FUNCTION_BLOCK FB_RobotRegionMove_FeedInConveyor_V2 EXTENDS FB_ObjectBase_V2 IMPLEMENTS IBasicElement
VAR_INPUT
    Robot     					: REFERENCE TO FB_FanucRobot_Basic_V2;
	LowerConveyor				: REFERENCE TO FB_Motor;
	Input 						: REFERENCE TO ST_InputTable;

   // Command   : ST_WareHouseWithRobotMove_Command;
    Info	  					: ST_RobotRegionMove_Info;
	Stop	  					: BOOL;
	bCheckUpperCV_ServiceDone	: BOOL;
END_VAR
VAR_OUTPUT
  // Status : ST_WareHouseWithRobotMove_Status;
  
END_VAR
VAR
	//_Abort		: BOOL;
	strStatus	: STRING;
	uiResumeStep : UDINT;
	
	Area	: E_RobotArea := E_RobotArea.InOutConveyor;
	UseA 	: BOOL;
	UseB	: BOOL;
	
	Get 	:BOOL;
	tonTimeOut	:TON;
	bTimeOutIN			   : BOOL;
	tonDelay	 : TON;
	_UniqueErrorCode :STRING;
	PreviousStrStatus : STRING;
	PreviousErrorCode : STRING;
	//Added by Jidien Kachu in 2025/10/09
	uiLastBothStep	: UINT;
	uiLastSingleClampStep	: UINT;
	bRobotTimeOutIN	: BOOL;
	tonRobotTimeOut	: TON;
	uiBothStep	: UINT;
	uiSingleClampStep	: UINT;	
	
	_bRetry	: BOOL;
END_VAR

SUPER^.A10_StateControl();
A00_BasicUnits();

(*============================================================
Create Date : 2025/11/24
Last Update	: 2026/04/01
Change Log  : 2025/11/24，Fix StateControl Switch , the version extend Kachue verion from TH_Mirror DAS // Edited : Gamin
			  2026/04/01，移植泰興鏡射機版本。
============================================================*)

ACTION A00_BasicUnits:
tonTimeOut(IN:= bTimeOutIN AND NOT THIS^.Stop, PT:=T#60S);
tonDelay(PT:=T#1S);
tonRobotTimeOut(IN:= bRobotTimeOutIN AND NOT THIS^.Stop, PT:=T#60S);
ErrorID:=2240;
END_ACTION

METHOD M_CheckCommand : BOOL // True : Command is useful
VAR_INPUT
END_VAR
VAR
	
END_VAR
// Check command paremeter is correct
	
	THIS^.Get :=Info.Get;
	UseA := Info.UseA;
	UseB := Info.UseB;

	 //FeedIn/Out conveyor
	 	IF UseA THEN	 
			IF  (Info.A_Position<1 OR  Info.A_Position>3 )THEN
				strStatus:='Wrong command ,Position A Not allow';
				M_CheckCommand:=FALSE;
				RETURN;	
			ELSIF  Info.A_Position=3 AND Get THEN
				strStatus:='Wrong command ,Can Not Get box from FeedOut conveyor ';
				M_CheckCommand:=FALSE;
				RETURN;
			ELSIF 	Info.A_Position <>3 AND NOT Get THEN
				strStatus:='Wrong command ,Can Not Put box to FeedIn conveyor ';
				M_CheckCommand:=FALSE;
				RETURN;				
			END_IF
		END_IF
		
		IF UseB AND ( Info.B_Position<1 OR  Info.B_Position>3 )THEN
			strStatus:='Wrong command ,Position B Not allow';
			M_CheckCommand:=FALSE;
			RETURN;	
		ELSIF UseB AND Info.B_Position=3 AND Get THEN
			strStatus:='Wrong command ,Can Not Get box from FeedOut conveyor ';
			M_CheckCommand:=FALSE;
			RETURN;		
		ELSIF UseB AND Info.B_Position <>3 AND NOT Get THEN
			strStatus:='Wrong command ,Can Not Put box to FeedIn conveyor ';
			M_CheckCommand:=FALSE;
			RETURN;		
		END_IF
		
M_CheckCommand:=TRUE;
END_METHOD

METHOD M_CheckUnitsNotBusy : BOOL
VAR_INPUT
END_VAR
M_CheckUnitsNotBusy := true;
END_METHOD

METHOD M_CheckUnitsReady : BOOL
VAR_INPUT
END_VAR
M_CheckUnitsReady := true;
END_METHOD

METHOD M_ResetHomingFeedOut : BOOL
VAR_INPUT
END_VAR
Execute := FALSE;
info.UseA := FALSE;
info.UseB := FALSE;

M_ResetHomingFeedOut := TRUE;
END_METHOD

METHOD M_StartHomingFeedOut : BOOL
VAR_INPUT
	UseA	: BOOL;
	UseB	: BOOL;
END_VAR
// NG conveyor homing only place
Info.Get := FALSE;

Info.UseA := UseA;
info.UseB := UseB;

IF UseA AND UseB THEN
	Info.A_Position := 3;
	Info.B_Position := 3;
ELSIF UseA THEN
	Info.A_Position := 3;
	info.B_Position := 99;
ELSIF UseB THEN
	info.A_Position	:= 99;
	Info.B_Position := 3;
END_IF

Execute := TRUE;

M_StartHomingFeedOut := TRUE;
END_METHOD

METHOD  M_STATE_ABORTED
VAR_INPUT
END_VAR
IF NOT _bRetry THEN
	Busy	:= FALSE;
	Error 	:= TRUE;
	Aborted := TRUE;
	Status 	:= strStatus;
	UniqueErrorCode:=_UniqueErrorCode;
	uiAbortingStep := 0;
	_AbortCompleted:=FALSE;//Edited by Jidien Kachu in 2025/10/14
END_IF

IF reset THEN
	_bRetry := TRUE;
	Error 	:= FALSE;
	Aborted := FALSE;
END_IF

IF NOT Execute THEN
	eSTATE:=STATE_RESETTING;
END_IF
IF Execute AND _bRetry AND NOT Robot._DI1.Error AND NOT Robot.Halt THEN
	PreviousStrStatus := strStatus;
	PreviousErrorCode := _UniqueErrorCode;
	uiExecutingStep   := uiResumeStep;
	(* Edited by Jidien Kachu in 2025/10/09 *)
	uiBothStep 		  := uiLastBothStep;
	uiSingleClampStep := uiLastSingleClampStep;

	Status := '';

	(*====================================*)
	IF GVL_ADS.MachineState <>E_MachineState.Error THEN
		eSTATE:=STATE_EXECUTING;
	END_IF
END_IF
END_METHOD

METHOD  M_STATE_ABORTING
VAR_INPUT
END_VAR
CASE uiAbortingStep OF
	0 :
			bTimeOutIN		:= FALSE;
			bRobotTimeOutIN := FALSE;
			tonDelay.IN 	:= FALSE;
			_bRetry:= FALSE;
			_Abort := FALSE;
			
			LowerConveyor.M_MotorStop();
			IF strStatus = PreviousStrStatus THEN
				_UniqueErrorCode :=PreviousErrorCode;
			END_IF
			uiAbortingStep:=100;
	100:		
			 IF DAS_CoreSys.MachineControl.M_RobotResetCmd() THEN
				 uiAbortingStep := 200;
			 END_IF
	200:
			IF DAS_CoreSys.MachineControl.M_RobotStartCmd() THEN
				 uiAbortingStep := 300;
			 END_IF 
	300:
			IF Robot._DI1.Error THEN
		 		uiAbortingStep := 100;
			ELSE
				uiAbortingStep := 9999;
			END_IF
	
	9999:	
			_AbortCompleted:=TRUE;
END_CASE

IF _AbortCompleted THEN	
	eSTATE :=STATE_ABORTED;
END_IF
END_METHOD

METHOD  M_STATE_DONE
VAR_INPUT
END_VAR
Busy := FALSE;
Done := TRUE;
IF NOT Execute THEN
    eState := STATE_RESETTING;
END_IF
END_METHOD

METHOD  M_STATE_DORMANT
VAR_INPUT
END_VAR
// Clear FB output
Busy            := FALSE;
Done            := FALSE;
_Abort			:= FALSE;
Aborted         := FALSE;
Error           := FALSE;
ErrorID         := 0;
Status          := '';
_ResetCompleted := FALSE;
_Error          := FALSE;
_Executed       := FALSE;
tonDelay.IN := FALSE;
bTimeOutIN:=FALSE;
bRobotTimeOutIN := FALSE;
strStatus :='No Error';
uiExecutingStep :=uiResettingStep :=uiResumeStep :=0;
uiBothStep			:= 0; 
uiSingleClampStep 	:= 0;
uiLastBothStep		:= 0; 
uiLastSingleClampStep := 0; 
_UniqueErrorCode :='0';
tonRobotTimeOut.IN := FALSE;
PreviousStrStatus			 :='';
PreviousErrorCode			 :='';
_bRetry				:= FALSE;

// Wait Execute command
IF Execute AND NOT stop THEN
    eState := STATE_EXECUTING;
END_IF
END_METHOD

METHOD  M_STATE_ERROR
VAR_INPUT
END_VAR
ERROR   :=TRUE;
Busy	:=FALSE;
Status := strStatus;
UniqueErrorCode:=_UniqueErrorCode;
IF NOT Execute THEN	
eSTATE:=STATE_RESETTING;
END_IF
END_METHOD

METHOD  M_STATE_EXECUTING
VAR_INPUT
END_VAR
VAR_INST
	BoxReady_1st : BOOL;
	BoxReady_2nd : BOOL;
//    uiBothStep : UINT;
//    uiSingleClampStep : UINT;	
	Address_A : INT;
	Address_B : INT;
END_VAR
VAR
	WareHouse: INT;
END_VAR
// Set Busy active edit by johnson
Busy := TRUE;
(*IF THIS^.Stop THEN // Pending the timeout when Stop signal occur
	bTimeoutIN:=FALSE;
END_IF*)
// Service Process
CASE uiExecutingStep OF
	0:
        // Clear variable
//        uiBothStep := 0;
		uiLastBothStep := 0; //Edited by Jidien Kachu in 2025/10/09
//		uiSingleClampStep :=0;
		uiLastSingleClampStep := 0; //Edited by Jidien Kachu in 2025/10/09
		BoxReady_1st := 0;
		BoxReady_2nd := 0;
		bTimeOutIN:=FALSE;
        // Check command
        IF M_CheckCommand() THEN
            uiExecutingStep := 10;
		ELSE
			_Error:=TRUE;
        END_IF
    10:
        // Start process, check units first
        IF M_CheckUnitsReady() THEN
            uiExecutingStep := 20;
        END_IF
    20:
        // CHeck units not busy state
        IF M_CheckUnitsNotBusy() THEN
            uiExecutingStep := 1000;
        END_IF
   
	1000:   
			// Read   coordinate
			 Area := THIS^.Area;
 			 Address_A := LREAL_TO_INT(Info.A_Position);
			 Address_B := LREAL_TO_INT(Info.B_Position);
			 
			IF UseA AND NOT UseB THEN
				//Only clampA
				uiExecutingStep := 10000;
			ELSIF NOT UseA AND UseB THEN
				//Only ClampB 
				uiExecutingStep := 20000;
			ELSIF UseA AND UseB THEN
				//Both Clamps
				uiExecutingStep := 30000;		
			ELSE
				strStatus := 'FB_RobotRegionMove_FeedInConveyor_V2 Step 1000: No clamp selected';
				_Error 	  := TRUE;
			END_IF

	10000:	// 檢查 A爪 Sensor判斷是否可以安全做動
			IF Get THEN
				IF  Robot._DI1.ClampA_Open THEN		// AClamp has box
					uiExecutingStep := 11000;
				ELSE
					_Error 	  := TRUE;
					strStatus := 'FB_RobotRegionMove_FeedInConveyor_V2 Step 10000: AClamp not open';
				END_IF
			ELSE
				IF NOT Robot._DI1.ClampA_Open THEN	// AClamp has box
					uiExecutingStep := 11000;
				ELSE	
					_Error 	  := TRUE;
					strStatus := 'FB_RobotRegionMove_FeedInConveyor_V2 Step 10000: AClamp is open';
				END_IF
			END_IF
       
    11000: // Only ClampA 
        IF NOT Robot._DI1.Done THEN
            
            
			CASE uiSingleClampStep OF
				
				0://
				
					CASE Address_A OF
						1,2:
							uiSingleClampStep:=1000;
						
						3: 
							uiSingleClampStep:=100;
					END_CASE
				
				100:	
					LowerConveyor.M_MoveBackward();
					tonDelay.IN := FALSE;
					IF ( NOT Input.bLowCV_BoxArrived_Sensor) AND ( Input.bLowCV_2ndBoxGap_Sensor) THEN
						bTimeOutIN:=FALSE;
						uiSingleClampStep:=150;
					END_IF
					bTimeOutIN:=TRUE;
					IF tonTimeOut.Q=TRUE OR Robot._DI1.Error THEN
						strStatus := 'FB_RobotRegionMove_FeedInConveyor_V2 Step 11000: Empty conveyor timeout';
						uiResumeStep:=11000;
						uiLastSingleClampStep := 0; //Edited by Jidien Kachu in 2025/10/09
						uiAbortingStep := 0;//Edited by Jidien Kachu in 2025/10/14
						_Abort:=TRUE;
					END_IF
				150:
					tonDelay.IN := TRUE;
					IF tonDelay.Q THEN
						uiSingleClampStep:=200;
					END_IF	
				200:
					tonDelay.IN := FALSE;
					LowerConveyor.M_MotorStop();
					uiSingleClampStep:=300;
				
				300:
					IF 	LowerConveyor.InStopped THEN
						bTimeOutIN:=FALSE;
						BoxReady_1st:=TRUE;
						uiSingleClampStep:=9999;
					END_IF
					bTimeOutIN:=TRUE;
					IF tonTimeOut.Q=TRUE OR Robot._DI1.Error THEN
						strStatus :='FB_RobotRegionMove_FeedInConveyor_V2 Step 11000: Stop Conveyor timeout';


						(* Edited by Jidien Kachu in 2025/10/09*)
//						_Error:=TRUE;
						uiResumeStep:=11000;
						uiLastSingleClampStep := 200;
						uiAbortingStep := 0;//Edited by Jidien Kachu in 2025/10/14
						_Abort:=TRUE;
						(*===================================*)
					END_IF	
				
				1000:
						CASE Address_A OF
						1:
								IF 	bCheckUpperCV_ServiceDone THEN
							BoxReady_1st:=Input.bUpCV_Block1Detect_Sensor;
								END_IF
						2:
								IF 	bCheckUpperCV_ServiceDone THEN
							BoxReady_1st:=Input.bUpCV_BoxArrived_Sensor;
								END_IF
						END_CASE						
						
				9999: //
						;
			END_CASE
			          		 
				  // Robot Abs move
           		 Robot.M_StartRobotAbsMove(GetBox:=Get,
											UseClampA:=UseA,
											UseClampB:=UseB,
											Area:=Area,
											ClampA_Address:=Address_A,
											ClampB_Address:=Address_B,
											BoxReady_1:=BoxReady_1st,
											BoxReady_2:=BoxReady_2nd);				  
		
        ELSE
//			bTimeOutIN:=FALSE;
			bRobotTimeOutIN := FALSE; //edited by Jidien Kachu in 2025/10/09
            uiExecutingStep := 10080;
        END_IF
		(* Edited by Jidien Kachu in 2025/10/09*)

		bRobotTimeOutIN := TRUE;

		IF tonRobotTimeOut.Q THEN

			bRobotTimeOutIN := FALSE;
			uiResumeStep 	:= 11000;
			strStatus 		:= 'FB_RobotRegionMove_FeedInConveyor_V2 Step 11000: Robot Abs move timeout';
			_Abort			:= TRUE;
		END_IF	
		IF Robot.Error THEN
			bRobotTimeOutIN := FALSE;
			uiResumeStep 	:= 11000;
			strStatus 		:= CONCAT('FB_RobotRegionMove_FeedInConveyor_V2',robot.ErrMsg);
			_Abort			:= TRUE;
		END_IF
		(*===================================*)
    10080:
        Robot.M_ResetRobotAbsMove(UseA,UseB); // Clear command and go to place box

		bRobotTimeOutIN := TRUE; //Edited by Jidien Kachu in 2025/10/09
        IF NOT Robot._DI1.Done THEN

			bRobotTimeOutIN := FALSE; //Edited by Jidien Kachu in 2025/10/09
            uiExecutingStep := 80000; 
        END_IF
		(* Edited by Jidien Kachu in 2025/10/09 *)

		IF tonRobotTimeOut.Q THEN
			bRobotTimeOutIN := FALSE;
			strStatus 		:= 'FB_RobotRegionMove_FeedInConveyor_V2 Step 10080: Reset Robot timeout';
			_Error:=TRUE;
		END_IF	
		(*=====================================*)
    
	10090: // Check box 

	20000:	// 檢查 B爪 Sensor判斷，是否可以安全做動。
			IF Get THEN
				IF  Robot._DI1.ClampB_Open THEN	// BClamp has box
					uiExecutingStep := 21000;
				ELSE
					_Error	  := TRUE;
					strStatus := 'FB_RobotRegionMove_FeedInConveyor_V2 Step 20000: BClamp not open';
				END_IF
			ELSE
				IF NOT Robot._DI1.ClampB_Open THEN	// BClamp has box
					uiExecutingStep := 21000;
				ELSE
					_Error	  := TRUE;
					strStatus := ' FB_RobotRegionMove_FeedInConveyor_V2 Step 20000: BClamp is open';
				END_IF
			END_IF
		
			
    21000: // Only ClampB
        IF NOT Robot._DI1.Done THEN
			
            	CASE uiSingleClampStep OF
				
				0://
				
					CASE Address_B OF
						1,2:
							uiSingleClampStep:=1000;
						
						3: 
							uiSingleClampStep:=100;
					END_CASE
			
				100:	
					LowerConveyor.M_MoveBackward();
					IF (NOT Input.bLowCV_BoxArrived_Sensor) AND  Input.bLowCV_2ndBoxGap_Sensor THEN
						bTimeOutIN:=FALSE;
						tonDelay.IN := FALSE;
						uiSingleClampStep:=150;
					END_IF
					bTimeOutIN:=TRUE;
					IF tonTimeOut.Q=TRUE OR Robot._DI1.Error THEN
						strStatus 				:= 'FB_RobotRegionMove_FeedInConveyor_V2 Step 21000: Empty conveyor timeout';
						uiResumeStep			:= 21000;
						uiLastSingleClampStep 	:= 0; //Edited by Jidien Kachu in 2025/10/09
						uiAbortingStep 			:= 0;//Edited by Jidien Kachu in 2025/10/14
						_Abort					:= TRUE;
					END_IF
					
				150:
					tonDelay.IN := TRUE;
					IF tonDelay.Q THEN
						uiSingleClampStep:=200;
					END_IF		
				200:
					tonDelay.IN := FALSE;
					LowerConveyor.M_MotorStop();
					uiSingleClampStep:=300;
				
				300:
					IF 	LowerConveyor.InStopped THEN
						bTimeOutIN:=FALSE;
						BoxReady_2nd:=TRUE;
						uiSingleClampStep:=9999;
					END_IF
					bTimeOutIN:=TRUE;
					IF tonTimeOut.Q=TRUE OR Robot._DI1.Error THEN
						strStatus :='FB_RobotRegionMove_FeedInConveyor_V2 Step 21000: Stop Conveyor timeout';




//						_Error:=TRUE;
						(* Edited by Jidien Kachu in 2025/10/09 *)
						uiResumeStep := 21000;
						uiLastSingleClampStep := 200;
						uiAbortingStep := 0;//Edited by Jidien Kachu in 2025/10/14
						_Abort := TRUE;
						(*====================================*)
					END_IF	
				
				1000:

						CASE Address_B OF
						1:
							IF 	bCheckUpperCV_ServiceDone THEN
								BoxReady_2nd:=Input.bUpCV_Block1Detect_Sensor;
							END_IF
													
						2:
							IF 	bCheckUpperCV_ServiceDone THEN
								BoxReady_2nd:=Input.bUpCV_BoxArrived_Sensor;
							END_IF

						END_CASE						
						
				9999 ://
			END_CASE	
		
			
			          		 
				  // Robot Abs move
           		 Robot.M_StartRobotAbsMove( GetBox:=Get,
											UseClampA:=UseA,
											UseClampB:=UseB,
											Area:=Area,
											ClampA_Address:=Address_A,
											ClampB_Address:=Address_B,
											BoxReady_1:=BoxReady_1st,
											BoxReady_2:=BoxReady_2nd);	
        ELSE
//			bTimeOutIN:=FALSE;
			bRobotTimeOutIN := FALSE; //Edited by Jidien Kachu in 2025/10/09
            uiExecutingStep := 20080;
        END_IF
		(* Edited by Jidien Kachu in 2025/10/09 *)

		bRobotTimeOutIN := TRUE;

		IF tonRobotTimeOut.Q THEN

			bRobotTimeOutIN := FALSE;
			uiResumeStep 	:= 21000;
			strStatus 		:= 'FB_RobotRegionMove_FeedInConveyor_V2 Step 21000: Robot Abs move timeout';
			_Abort			:= TRUE;
		END_IF	
		IF Robot.Error THEN
			bRobotTimeOutIN := FALSE;
			uiResumeStep 	:= 21000;
			strStatus 		:= CONCAT('FB_RobotRegionMove_FeedInConveyor_V2',robot.ErrMsg);
			_Abort			:= TRUE;
		END_IF
		(*====================================*)
    20080:
       Robot.M_ResetRobotAbsMove(UseA,UseB);; // Clear command 

        IF NOT Robot._DI1.Done THEN
			bRobotTimeOutIN := FALSE; // Edited by Jidien Kachu in 2025/10/09
            uiExecutingStep := 80000; 
        END_IF
		(* Edited by Jidien Kachu in 2025/10/09 *)

		bRobotTimeOutIN := TRUE;

		IF tonRobotTimeOut.Q THEN
			bRobotTimeOutIN := FALSE;
			strStatus :='FB_RobotRegionMove_FeedInConveyor_V2 Step 20080: Reset Robot timeout';


			_Error:=TRUE;
		END_IF	
		(*===================================*)
	
	30000:
			IF Get THEN
				IF   Robot._DI1.ClampA_Open AND Robot._DI1.ClampB_Open THEN
					uiExecutingStep := 31000;
				ELSE
					_Error	  := TRUE;
					strStatus := 'FB_RobotRegionMove_FeedInConveyor_V2 Step 30000: Clamp not open';
				END_IF
			ELSE
				IF NOT Robot._DI1.ClampA_Open AND NOT Robot._DI1.ClampB_Open THEN
					uiExecutingStep := 31000;
				ELSE
					_Error	  := TRUE;
					strStatus := 'FB_RobotRegionMove_FeedInConveyor_V2 Step 30000: Clamp is open';
				END_IF 
			END_IF		
		
		
    31000: // Both Clamps
        		
		
		  CASE uiBothStep OF
           		0://	
					BoxReady_1st := FALSE;
					BoxReady_2nd := FALSE;
					CASE Address_A OF
						1,2:
							uiBothStep:=1000;
						
						3: 
							uiBothStep:=100;
					END_CASE				
				100:	
					tonDelay.IN := FALSE;
					LowerConveyor.M_MoveBackward();
					bTimeOutIN:=FALSE;
					IF (NOT Input.bLowCV_BoxArrived_Sensor) AND  Input.bLowCV_2ndBoxGap_Sensor THEN
						uiBothStep:=150;
					END_IF
					bTimeOutIN:=TRUE;
					IF tonTimeOut.Q=TRUE OR Robot._DI1.Error THEN
						strStatus 		:= 'FB_RobotRegionMove_FeedInConveyor_V2 Step 31000: Empty conveyor timeout';
						Error 			:= TRUE;
						uiResumeStep	:= 31000;
						uiLastBothStep  := 0; //Edited by Jidien Kachu in 2025/10/09
						uiAbortingStep  := 0;//Edited by Jidien Kachu in 2025/10/14
						_Abort:=TRUE;
					END_IF	
					
				150:
					tonDelay.IN := TRUE;
					IF tonDelay.Q THEN
						uiBothStep:=200;
					END_IF		
				200:
					tonDelay.IN := FALSE;
					LowerConveyor.M_MotorStop();
					uiBothStep:=300;
				
				300:
					IF 	LowerConveyor.InStopped THEN
						bTimeOutIN:=FALSE;
						BoxReady_1st:=TRUE;
						uiBothStep:=1000;
					END_IF
					bTimeOutIN:=TRUE;
					IF tonTimeOut.Q=TRUE OR Robot._DI1.Error THEN
						strStatus :='FB_RobotRegionMove_FeedInConveyor_V2 Step 31000: Stop conveyor timeout';




						(* Edited by Jidien Kachu in 2025/10/09 *)
//						_Error:=TRUE;
						uiResumeStep := 31000;
						uiLastBothStep := 200;
						uiAbortingStep := 0;//Edited by Jidien Kachu in 2025/10/14
						_Abort := TRUE;
						(*====================================*)
					END_IF		

				1000:
							CASE Address_A OF							
						1:
								IF bCheckUpperCV_ServiceDone THEN
							BoxReady_1st:=Input.bUpCV_Block1Detect_Sensor;
								END_IF
						2:
								IF bCheckUpperCV_ServiceDone THEN
							BoxReady_1st:=Input.bUpCV_BoxArrived_Sensor;
								END_IF
						END_CASE
						



						IF Robot._DI1.Notification THEN

							uiBothStep:=2000;
						END_IF
						
						
				2000:

						CASE Address_B OF
						1,2:
							uiBothStep:=9000;						
						3: 
							uiBothStep:=3000;
					END_CASE	
				
				3000:	
					tonDelay.IN := FALSE;
					LowerConveyor.M_MoveBackward();
					IF (NOT Input.bLowCV_BoxArrived_Sensor) AND Input.bLowCV_2ndBoxGap_Sensor THEN
						bTimeOutIN:=FALSE;
						uiBothStep:=3100;
					END_IF
					bTimeOutIN:=TRUE;
					IF tonTimeOut.Q=TRUE OR Robot._DI1.Error THEN
						strStatus := 'FB_RobotRegionMove_FeedInConveyor_V2 Step 31000: Empty conveyor timeout';
						uiResumeStep:=31000;
						uiLastBothStep := 2000; // Edited by Jidien Kachu in 2025/10/09
						uiAbortingStep := 0;//Edited by Jidien Kachu in 2025/10/14
						_Abort:=TRUE;
					END_IF	
					
				3100:
					
					tonDelay.IN := TRUE;
					IF tonDelay.Q THEN
						uiBothStep:=3200;
					END_IF		
				3200:
					tonDelay.IN := FALSE;
					LowerConveyor.M_MotorStop();
					uiBothStep:=3300;
				
				3300:
					IF 	LowerConveyor.InStopped THEN
						bTimeOutIN:=FALSE;
						BoxReady_2nd:=TRUE;
						uiBothStep:=9999;
					END_IF
					bTimeOutIN:=TRUE;
					IF tonTimeOut.Q=TRUE OR Robot._DI1.Error THEN
						strStatus :='FB_RobotRegionMove_FeedInConveyor_V2 Step 31000: Stop conveyor timeout';




						(* Edited by Jidien Kachu in 2025/10/09 *)
//						_Error:=TRUE;
						uiResumeStep := 31000;
						uiLastBothStep := 3200;
						uiAbortingStep := 0;//Edited by Jidien Kachu in 2025/10/14
						_Abort := TRUE;
						(*====================================*)
					END_IF		
				9000:
							CASE Address_B OF							
						1:
								IF bCheckUpperCV_ServiceDone THEN
									BoxReady_2nd:=Input.bUpCV_Block1Detect_Sensor;
								END_IF
						
						2:
								IF bCheckUpperCV_ServiceDone THEN
							BoxReady_2nd:=Input.bUpCV_BoxArrived_Sensor;
								END_IF

						END_CASE
				
				9999: //Wait		
        // wait reset
        END_CASE

       	  // Robot Abs move
           		 Robot.M_StartRobotAbsMove( GetBox:=Get,
											UseClampA:=UseA,
											UseClampB:=UseB,
											Area:=Area,
											ClampA_Address:=Address_A,
											ClampB_Address:=Address_B,
											BoxReady_1:=BoxReady_1st,
											BoxReady_2:=BoxReady_2nd);	
		
		
        IF Robot._DI1.Done THEN

			bRobotTimeOutIN := FALSE; //Edited by Jidien Kachu in 2025/10/09
            uiExecutingStep := 30080;
        END_IF
		(* Edited by Jidien Kachu in 2025/10/09*)

		bRobotTimeOutIN := TRUE;

		IF tonRobotTimeOut.Q THEN

			bRobotTimeOutIN := FALSE;
			uiResumeStep	:= 31000;
		(*===================================*)
			strStatus := 'FB_RobotRegionMove_FeedInConveyor_V2 Step 31000: Robot Abs move timeout'; 
			_Abort			:= TRUE;
		END_IF
		IF Robot.Error THEN
			bRobotTimeOutIN	:= FALSE;
			uiResumeStep	:= 31000;
			strStatus		:= CONCAT('FB_RobotRegionMove_FeedInConveyor_V2',robot.ErrMsg);
			_Abort			:= TRUE;
		END_IF
    30080: // Check robot command is clear
        
        Robot.M_ResetRobotAbsMove(UseA,UseB);

        IF NOT Robot._DI1.Done THEN
			(* Edited by Jidien Kachu in 2025/10/09*)

			bRobotTimeOutIN := FALSE;
            uiExecutingStep := 80000; // go to place step
        END_IF    

		bRobotTimeOutIN := TRUE;

		IF tonRobotTimeOut.Q THEN
			(*===================================*)
			strStatus :='FB_RobotRegionMove_FeedInConveyor_V2 Step 31080: Stop Robot timeout';


			_Error:=TRUE;
		END_IF	
   
		
	80000:
		IF UseA THEN
			CASE Address_A OF
			1:
//				IF Input.bUpCV_BoxArrived_Sensor.P_SignalState THEN
//					strStatus :='Box not taken on F1';
//					_Error:=TRUE;
//				END_IF
				 uiExecutingStep :=99000;
			2:	
//				IF Input.bUpCV_Block1Detect_Sensor.P_SignalState THEN
//					strStatus :='Box not taken on F2';
//					_Error:=TRUE;
//				END_IF	
					uiExecutingStep :=99000;

			3:
				uiExecutingStep :=81000;			
			END_CASE
		END_IF
		IF UseB THEN
			CASE Address_B OF
			1:
//				IF Input.bUpCV_BoxArrived_Sensor.P_SignalState THEN
//					strStatus :='Box not taken on F1';
//					_Error:=TRUE;
//				END_IF
				 uiExecutingStep :=99000;
			2:	
//				IF Input.bUpCV_Block1Detect_Sensor.P_SignalState THEN
//					strStatus :='Box not taken on F2';
//					_Error:=TRUE;
//				END_IF	
					uiExecutingStep :=99000;

			3:
				uiExecutingStep :=81000;			
			END_CASE
		END_IF
		
	81000:
			LowerConveyor.M_MoveBackward();
			bTimeOutIN:=FALSE;
			IF (NOT Input.bLowCV_BoxArrived_Sensor) AND ( Input.bLowCV_2ndBoxGap_Sensor) THEN
						uiExecutingStep:=81100;
			END_IF
			bTimeOutIN:=TRUE;
			IF tonTimeOut.Q=TRUE OR Robot._DI1.Error THEN
				strStatus :='FB_RobotRegionMove_FeedInConveyor_V2 Step 81000: Empty conveyor timeout';


				(* Edited by Jidien Kachu in 2025/10/09 *)

				uiResumeStep := 81000;
				uiAbortingStep := 0;//Edited by Jidien Kachu in 2025/10/14
				_Abort := TRUE;
				(*====================================*)
			END_IF	
	81100:		
			LowerConveyor.M_MotorStop();
			uiExecutingStep:=81200;
				
	81200:
			IF 	LowerConveyor.InStopped THEN
				bTimeOutIN:=FALSE;
				uiExecutingStep:=99000;
			END_IF
			bTimeOutIN:=TRUE;
			IF tonTimeOut.Q=TRUE OR Robot._DI1.Error THEN
				strStatus :='FB_RobotRegionMove_FeedInConveyor_V2 Step 81200: Stop conveyor timeout';


				(* Edited by Jidien Kachu in 2025/10/09 *)

				uiResumeStep := 81100;
				uiAbortingStep := 0;//Edited by Jidien Kachu in 2025/10/14
				_Abort := TRUE;
				(*====================================*)
			END_IF		
					
    99000: 	  // process done
          Status    := 'Process completed';
      	  _Executed := TRUE;
		  uiBothStep:= 0; //Edited by Jidien Kachu in 2025/10/14
		  uiSingleClampStep := 0;//Edited by Jidien Kachu in 2025/10/14
END_CASE

// ================= STATE Control ==================
IF NOT Execute THEN
    eState 	:= STATE_RESETTING;
ELSIF _Error THEN
    eState	:= STATE_ERROR;
ELSIF _Abort THEN
	eSTATE	:= STATE_ABORTING;
ELSIF _Executed THEN
    eState 					:= STATE_DONE;
	uiLastBothStep 			:= 0; //Edited by Jidien Kachu in 2025/10/14
	uiLastSingleClampStep 	:= 0; //Edited by Jidien Kachu in 2025/10/14
END_IF
END_METHOD

METHOD  M_STATE_RESETTING
VAR_INPUT
END_VAR
Error :=FALSE;
Done :=FALSE;
Busy := FALSE;


CASE uiResettingStep OF
	
	0:
		tonDelay.IN := FALSE;
		bTimeOutIN:=FALSE;
		Robot.M_ResetAllCommand();
		Robot.M_ResetRobotAbsMove(TRUE,TRUE);
		uiResettingStep:=100;
		tonRobotTimeOut.IN := FALSE;
		
	100:
	
		LowerConveyor.M_MotorStop();	
		uiResettingStep:=9999;
	9999:
		_ResetCompleted:=TRUE;
END_CASE
IF _ResetCompleted THEN
	eSTATE:=STATE_DORMANT;
END_IF
END_METHOD

END_FUNCTION_BLOCK

(* stored: Version 1.1.0.1, ProductVersion 3.1.4024.13
   POU FB_RobotRegionMove_FeedInConveyor_V2: Id {6d0a658e-26e9-428a-8fcb-77a9287fbf35}, SpecialFunc None
   Folder Method: Id {6305d260-f295-4065-8899-9548086c506e}
   Folder State: Id {716f6113-c46b-4f3a-b90c-992391c0593c}
   Action A00_BasicUnits: Id {74e70b97-15e2-49e1-b024-58acfa896b23}
   Method M_CheckCommand: Id {7c9e136d-336c-4051-9f78-cb6d9d41ebb8}
   Method M_CheckUnitsNotBusy: Id {2a0a8711-20be-4879-808b-3059a1b196d8}
   Method M_CheckUnitsReady: Id {7e6121c5-899a-440b-aa4e-3e68caaca88d}
   Method M_ResetHomingFeedOut: Id {a5a2e305-1ffe-467c-a2c1-4b50b023570d}
   Method M_StartHomingFeedOut: Id {e41562bd-df64-4d10-8da3-66aed675428e}
   Method M_STATE_ABORTED: Id {47aa7add-804c-4c5c-ab3a-fbb5ffc5f469}
   Method M_STATE_ABORTING: Id {011f7f09-bffb-4bf5-a774-7d38be4067ad}
   Method M_STATE_DONE: Id {5832e808-21d5-474d-b38f-8763a4e2c532}
   Method M_STATE_DORMANT: Id {4f3197e5-279e-4441-859d-95aeaa87a794}
   Method M_STATE_ERROR: Id {9415c378-2d37-48ae-b43d-f37c5d76b2b1}
   Method M_STATE_EXECUTING: Id {5d3cdb97-d028-4fe6-b780-1ee84c62585a}
   Method M_STATE_RESETTING: Id {bfe90e01-7c06-4ede-9edd-d31754e1c84f} *)
